FUNCTION_BLOCK ABSTRACT FB_HMIInputBase //Base function for HMI inputs
VAR_INPUT
	bEnable : BOOL := TRUE ;
END_VAR
VAR_OUTPUT
	bInVisible			: BOOL := TRUE ; // input is visible (standard := NOT bEnable )
	bDeactivateInput	: BOOL := TRUE ; // input is enabled (Standard := bEnable)
END_VAR
VAR
END_VAR

SetHMIInstructions();

METHOD INTERNAL SetHMIInstructions : BOOL
VAR_INPUT
END_VAR
bInVisible 			:= NOT bEnable ;
bDeactivateInput	:= NOT bEnable ;
END_METHOD

METHOD ABSTRACT SetOutputToPLC : BOOL
VAR_INPUT
END_VAR
END_METHOD

END_FUNCTION_BLOCK

(* stored: Version 1.1.0.1, ProductVersion 3.1.4024.11
   POU FB_HMIInputBase: Id {9b228d30-0c34-4ec7-a1ab-f9487cc3d5ce}, SpecialFunc None
   Method SetHMIInstructions: Id {5dde2b73-b2f9-4ff5-b140-bb01c00a0aba}
   Method SetOutputToPLC: Id {4dfd4d0d-afb6-4187-8cbc-5a4339412b11} *)
